PROGRAM C13_CheckDuplicatesCACData
VAR
	fbCaseDuplicatCheck		: FB_CASE_DuplicatCheck;
	fbDuplicateUpdateToDB	: FB_CASE_DuplicateUpdateToDB;
	
	nOACFilesBlocked		: UINT;
	nOCVFilesBlocked		: UINT;
	stDaigOACDataDB				: ST_DB_OACDataCtrl;
	stDiagOCVDataDB				: ST_DB_OCVDataCtrl;
END_VAR

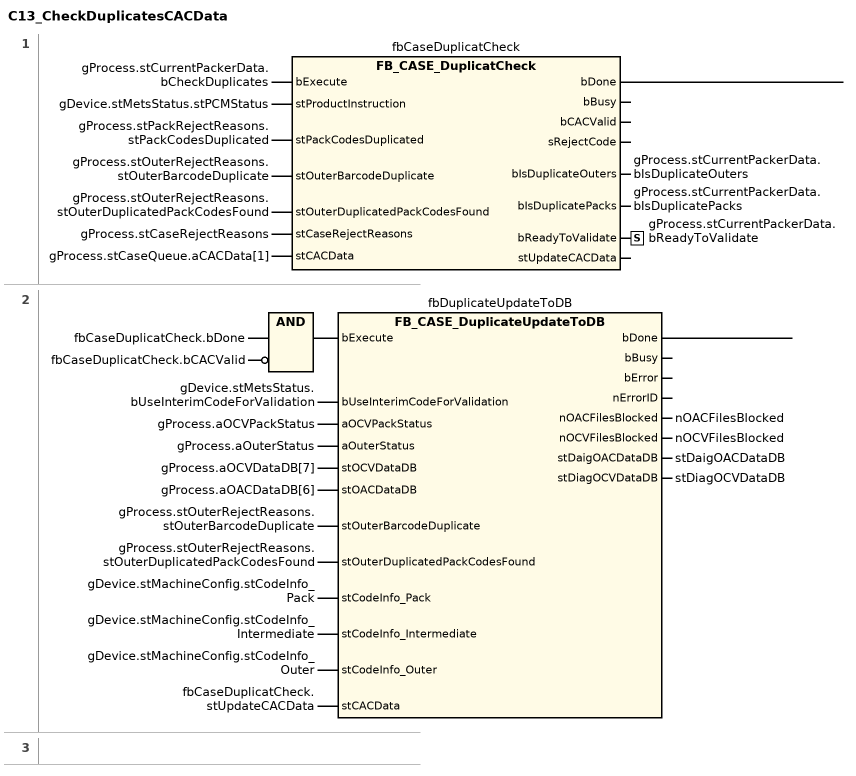
// NETWORK 1
fbCaseDuplicatCheck(
    bExecute := gProcess.stCurrentPackerData.bCheckDuplicates,
    stProductInstruction := gDevice.stMetsStatus.stPCMStatus,
    stPackCodesDuplicated := gProcess.stPackRejectReasons.stPackCodesDuplicated,
    stOuterBarcodeDuplicate := gProcess.stOuterRejectReasons.stOuterBarcodeDuplicate,
    stOuterDuplicatedPackCodesFound := gProcess.stOuterRejectReasons.stOuterDuplicatedPackCodesFound,
    stCaseRejectReasons := gProcess.stCaseRejectReasons,
    stCACData := gProcess.stCaseQueue.aCACData[1],
    bIsDuplicateOuters => gProcess.stCurrentPackerData.bIsDuplicateOuters,
    bIsDuplicatePacks => gProcess.stCurrentPackerData.bIsDuplicatePacks); // FB_CASE_DuplicatCheck
gProcess.stCurrentPackerData.bReadyToValidate S= fbCaseDuplicatCheck.bReadyToValidate;

// NETWORK 2
fbDuplicateUpdateToDB(
    bExecute := fbCaseDuplicatCheck.bDone AND NOT fbCaseDuplicatCheck.bCACValid,
    bUseInterimCodeForValidation := gDevice.stMetsStatus.bUseInterimCodeForValidation,
    aOCVPackStatus := gProcess.aOCVPackStatus,
    aOuterStatus := gProcess.aOuterStatus,
    stOCVDataDB := gProcess.aOCVDataDB[7],
    stOACDataDB := gProcess.aOACDataDB[6],
    stOuterBarcodeDuplicate := gProcess.stOuterRejectReasons.stOuterBarcodeDuplicate,
    stOuterDuplicatedPackCodesFound := gProcess.stOuterRejectReasons.stOuterDuplicatedPackCodesFound,
    stCodeInfo_Pack := gDevice.stMachineConfig.stCodeInfo_Pack,
    stCodeInfo_Intermediate := gDevice.stMachineConfig.stCodeInfo_Intermediate,
    stCodeInfo_Outer := gDevice.stMachineConfig.stCodeInfo_Outer,
    stCACData := fbCaseDuplicatCheck.stUpdateCACData,
    nOACFilesBlocked => nOACFilesBlocked,
    nOCVFilesBlocked => nOCVFilesBlocked,
    stDaigOACDataDB => stDaigOACDataDB,
    stDiagOCVDataDB => stDiagOCVDataDB); // FB_CASE_DuplicateUpdateToDB

// NETWORK 3

END_PROGRAM

(* stored: Version 1.1.0.1
   POU C13_CheckDuplicatesCACData: Id {e8f2d8b8-cb30-47ea-9986-f636535d9e7d}, SpecialFunc None *)
